{attribute 'GeneratedUsingTerminal: EL5001-0011-0019'}
{attribute addProperty BoxType "EL5001-0011-0019"}
{attribute addProperty Id "Data_errorBOOL1Frame_errorBOOL1Power_failureBOOL1TxPDO_StateBOOL1TxPDO_ToggleBOOL1"}
{attribute addProperty CRC "1399219146"}
{attribute addProperty Size "5"}
TYPE Status_536663CA :
STRUCT
	{attribute addProperty Name "Data_error"}
	Data_error : BOOL;
	{attribute addProperty Name "Frame_error"}
	Frame_error : BOOL;
	{attribute addProperty Name "Power_failure"}
	Power_failure : BOOL;
	{attribute addProperty Name "TxPDO_State"}
	TxPDO_State : BOOL;
	{attribute addProperty Name "TxPDO_Toggle"}
	TxPDO_Toggle : BOOL;
END_STRUCT
END_TYPE

(* stored: Version 1.2.0.0, ProductVersion 3.1.4024.9
   DUT Status_536663CA: Id {95e15b06-ae03-4374-97d1-12eefdff6091} *)
